PROGRAM branch2
VAR
END_VAR

END_PROGRAM

(* stored: Version 1.1.0.1, ProductVersion 3.1.4024.12
   POU branch2: Id {0bb389dd-2447-041b-0c77-c9844855d835}, SpecialFunc None *)
